(* PLC project Scenario_10, Beckhoff Automation GmbH TwinCAT PLC Control 3.5.8.40 *)
(* stored: creationDateTime 2017-05-02T11:08:00.4328535, modificationDateTime 2017-05-02T11:08:00.4378537 *)

PROGRAM MAIN
VAR		
	PPU : PPU;

//WPType	
	//Stack WPType
	Stack_WPType_Black : BOOL;
	Stack_WPType_White : BOOL;
	Stack_WPType_Metallic : BOOL;
	//Crane WPType
	Crane_WPType_Black : BOOL;
	Crane_WPType_White : BOOL;
	Crane_WPType_Metallic : BOOL;
	//Stamp WPType
	Stamp_WPType_Black : BOOL;
	Stamp_WPType_White : BOOL;
	Stamp_WPType_Metallic : BOOL;
	
//Free Signale for follow plant section
	//Stack
	Stack_WPProvided : BOOL;
	//Crane
	Crane_Allow_Conveyor_to_Operate : BOOL;
	Crane_Allow_Stamp_to_Operate : BOOL;
	Crane_PickedUpStackWP : BOOL;
	//Stamp	
	Stamp_IsStamping : BOOL;
	Stamp_WPAvailable : BOOL;
	Stamp_AutomaticExecuteCompleted	: BOOL;
	//Conveyor
	LargeSortingConveyor_AllowedToOperate : BOOL;
	LargeSortingConveyor_IsSorting : BOOL;
	LargeSortingConveyor_AutomaticExecuteCompleted : BOOL;
	
END_VAR

                  PPU();
PPU.Stack();
PPU.Crane();
PPU.Stamp();
PPU.LargeSortingConveyor();

//WPType
	//Stack WPType
	Stack_WPType_Black := PPU.Stack.WPType_Black;
	Stack_WPType_White := PPU.Stack.WPType_White;
	Stack_WPType_Metallic := PPU.Stack.WPType_Metallic;
	//Crane WPType
	Crane_WPType_Black := PPU.Crane.WPType_Black;
	Crane_WPType_White := PPU.Crane.WPType_White;
	Crane_WPType_Metallic := PPU.Crane.WPType_Metallic;
	//Stamp WPType
	Stamp_WPType_Black := PPU.Stamp.WPType_Black;
	Stamp_WPType_White := PPU.Stamp.WPType_White;
	Stamp_WPType_Metallic := PPU.Stamp.WPType_Metallic;
	
//Free Signale for follow plant section
	//Stack
	Stack_WPProvided := PPU.Stack.WPProvided;
	//Crane
	Crane_Allow_Conveyor_to_Operate := PPU.Crane.Conveyor_AllowedToOperate;
	Crane_Allow_Stamp_to_Operate := PPU.Crane.Stamp_AllowedToOperate;
	Crane_PickedUpStackWP := PPU.Crane.Table.AtStack.DI_SwitchTrue AND PPU.Crane.WPPickedUp;
	//Stamp
	Stamp_IsStamping := PPU.Stamp.IsStamping;
	Stamp_WPAvailable := PPU.Stamp.WPAvailable.DI_SwitchTrue;	
	Stamp_AutomaticExecuteCompleted := PPU.Stamp.AutomaticExecuteCompleted;
	//Conveyor
	LargeSortingConveyor_AllowedToOperate := Crane_Allow_Conveyor_to_Operate;
	LargeSortingConveyor_IsSorting := PPU.LargeSortingConveyor.IsSorting;
	LargeSortingConveyor_AutomaticExecuteCompleted := PPU.LargeSortingConveyor.AutomaticExecuteCompleted;
                
END_PROGRAM

FUNCTION_BLOCK BistableCylinder
VAR_INPUT	
END_VAR
VAR_OUTPUT
END_VAR
VAR	
	//Hardware
	DI_Extended AT %I* : BOOL;
	DI_Retracted AT %I* : BOOL;	
	DO_Extend AT %Q* : BOOL;
	DO_Retract AT %Q* : BOOL;
	//Software
	Extended : BOOL;
	Retracted : BOOL;
END_VAR

                  
                

ACTION ACT_Extend:
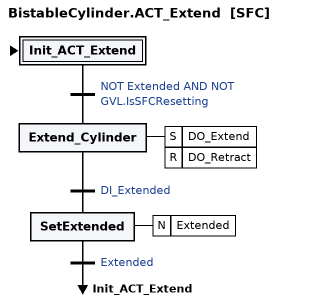
INITIAL_STEP Init_ACT_Extend:
END_STEP
TRANSITION FROM Init_ACT_Extend TO Extend_Cylinder
  := NOT Extended AND NOT GVL.IsSFCResetting;
END_TRANSITION
STEP Extend_Cylinder:
  DO_Extend(S);
  DO_Retract(R);
END_STEP
TRANSITION FROM Extend_Cylinder TO SetExtended
  := DI_Extended;
END_TRANSITION
STEP SetExtended:
  Extended(N);
END_STEP
TRANSITION FROM SetExtended TO Init_ACT_Extend
  := Extended;
END_TRANSITION
END_ACTION

ACTION ACT_Retract:
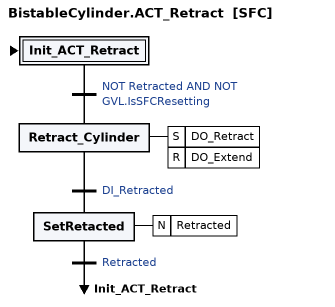
INITIAL_STEP Init_ACT_Retract:
END_STEP
TRANSITION FROM Init_ACT_Retract TO Retract_Cylinder
  := NOT Retracted AND NOT GVL.IsSFCResetting;
END_TRANSITION
STEP Retract_Cylinder:
  DO_Retract(S);
  DO_Extend(R);
END_STEP
TRANSITION FROM Retract_Cylinder TO SetRetacted
  := DI_Retracted;
END_TRANSITION
STEP SetRetacted:
  Retracted(N);
END_STEP
TRANSITION FROM SetRetacted TO Init_ACT_Retract
  := Retracted;
END_TRANSITION
END_ACTION
END_FUNCTION_BLOCK

FUNCTION_BLOCK InductiveSensor
VAR_INPUT
END_VAR
VAR_OUTPUT
END_VAR
VAR
	//Hardware
	DI_WPMetallic AT %I* : BOOL;
END_VAR

                  
                
END_FUNCTION_BLOCK

FUNCTION_BLOCK MicroSwitch
VAR_INPUT
END_VAR
VAR_OUTPUT
END_VAR
VAR
	//Hardware
	DI_SwitchTrue AT %I* : BOOL;
END_VAR

                  
                
END_FUNCTION_BLOCK

FUNCTION_BLOCK MonostableCylinder
VAR_INPUT	
END_VAR	
VAR_OUTPUT	
END_VAR
VAR	
	//Hardware
	DI_Extended AT %I* : BOOL;
	DI_Retracted AT %I* : BOOL;	
	DO_Extend AT %Q* : BOOL;
	//Software
	Extended : BOOL;
	Retracted : BOOL;
END_VAR

                  
                

ACTION ACT_Extend:
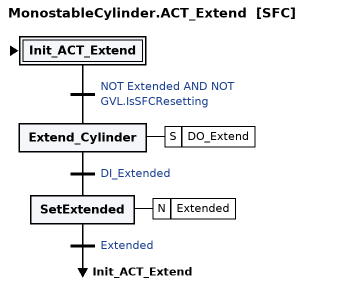
INITIAL_STEP Init_ACT_Extend:
END_STEP
TRANSITION FROM Init_ACT_Extend TO Extend_Cylinder
  := NOT Extended AND NOT GVL.IsSFCResetting;
END_TRANSITION
STEP Extend_Cylinder:
  DO_Extend(S);
END_STEP
TRANSITION FROM Extend_Cylinder TO SetExtended
  := DI_Extended;
END_TRANSITION
STEP SetExtended:
  Extended(N);
END_STEP
TRANSITION FROM SetExtended TO Init_ACT_Extend
  := Extended;
END_TRANSITION
END_ACTION

ACTION ACT_Retract:
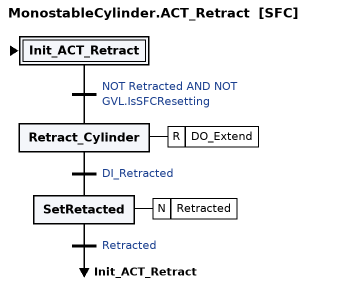
INITIAL_STEP Init_ACT_Retract:
END_STEP
TRANSITION FROM Init_ACT_Retract TO Retract_Cylinder
  := NOT Retracted AND NOT GVL.IsSFCResetting;
END_TRANSITION
STEP Retract_Cylinder:
  DO_Extend(R);
END_STEP
TRANSITION FROM Retract_Cylinder TO SetRetacted
  := DI_Retracted;
END_TRANSITION
STEP SetRetacted:
  Retracted(N);
END_STEP
TRANSITION FROM SetRetacted TO Init_ACT_Retract
  := Retracted;
END_TRANSITION
END_ACTION
END_FUNCTION_BLOCK

FUNCTION_BLOCK Motor
VAR_INPUT
END_VAR
VAR_OUTPUT	
END_VAR
VAR	
	//Hardware
	DO_TurnClockwise AT %Q* : BOOL;
	DO_TurnCounterclockwise AT %Q* : BOOL;
	//Software
	Stopped : BOOL;
	TurningClockwise : BOOL;
	TurningCounterclockwise : BOOL;
END_VAR

                  
                

ACTION ACT_Stop:
                      DO_TurnClockwise := FALSE;
DO_TurnCounterclockwise := FALSE;

Stopped := TRUE;
TurningClockwise := FALSE;
TurningCounterclockwise := FALSE;
                    
END_ACTION

ACTION ACT_TurnClockwise:
                      DO_TurnClockwise := TRUE;
DO_TurnCounterclockwise := FALSE;

Stopped := FALSE;
TurningClockwise := TRUE;
TurningCounterclockwise := FALSE;
                    
END_ACTION

ACTION ACT_TurnCounterclockwise:
                      DO_TurnClockwise := FALSE;
DO_TurnCounterclockwise := TRUE;

Stopped := FALSE;
TurningClockwise := FALSE;
TurningCounterclockwise := TRUE;
                    
END_ACTION
END_FUNCTION_BLOCK

FUNCTION_BLOCK OperationPanel
VAR_INPUT
END_VAR
VAR_OUTPUT
	//Software
	EmergencyStop : BOOL;
	StartButton : BOOL;
	ManuelMode : BOOL;
END_VAR
VAR
	//Hardware
	DI_StartButton AT %I* : BOOL;
	DI_ManuelButton AT %I* : BOOL;	
	DI_EmergencyStop AT %I* : BOOL;	
	DO_LampGreen AT %Q* : BOOL;
	DO_LampWhite AT %Q* : BOOL;
END_VAR

                  EmergencyStop := NOT DI_EmergencyStop;
StartButton := DI_StartButton;
ManuelMode := DI_ManuelButton;
                

ACTION ACT_TurnLampGreen_Off:
                      DO_LampGreen := FALSE;
                    
END_ACTION

ACTION ACT_TurnLampGreen_On:
                      DO_LampGreen := TRUE;
                    
END_ACTION

ACTION ACT_TurnLampWhite_Off:
                      DO_LampWhite:=FALSE;
                    
END_ACTION

ACTION ACT_TurnLampWhite_On:
                      DO_LampWhite:=TRUE;
                    
END_ACTION
END_FUNCTION_BLOCK

FUNCTION_BLOCK OpticalSensor
VAR_INPUT
END_VAR
VAR_OUTPUT
END_VAR
VAR
	//Hardware
	DI_WPLight AT %I* : BOOL;
END_VAR

                  
                
END_FUNCTION_BLOCK

FUNCTION_BLOCK PresenceSensor
VAR_INPUT
END_VAR
VAR_OUTPUT
END_VAR
VAR
	DI_WPDetected AT %I* : BOOL;
END_VAR

                  
                
END_FUNCTION_BLOCK

FUNCTION_BLOCK PressureSensor
VAR_INPUT
END_VAR
VAR_OUTPUT
END_VAR
VAR
	//Hardware
	AI_CurrentPressure AT %I* : INT;
END_VAR

                  
                
END_FUNCTION_BLOCK

FUNCTION_BLOCK ProportionalValve
VAR_INPUT
	//Hardware
	AO_SetPressure AT %Q* : INT;
END_VAR
VAR_OUTPUT
END_VAR
VAR	
END_VAR

                  
                
END_FUNCTION_BLOCK

FUNCTION_BLOCK TurningTable
VAR_INPUT
END_VAR
VAR_OUTPUT
END_VAR
VAR
	//Hardware
	Motor : Motor;
	AtStack : MicroSwitch;
	AtConveyor : MicroSwitch;
	AtStamp : MicroSwitch;
END_VAR

                  
                
END_FUNCTION_BLOCK

FUNCTION_BLOCK VacuumGripper
VAR_INPUT	
	//Hardware
	Valve : Valve;
	VacuumSwitch : VacuumSwitch;
END_VAR
VAR_OUTPUT	
END_VAR
VAR	
	//Software
	Intaken : BOOL;
	Released : BOOL;
END_VAR

                  
                

ACTION ACT_Intake:
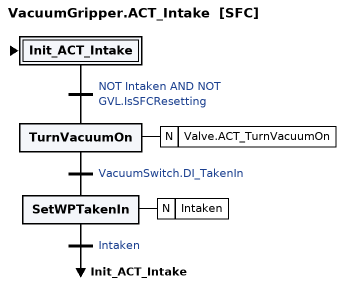
INITIAL_STEP Init_ACT_Intake:
END_STEP
TRANSITION FROM Init_ACT_Intake TO TurnVacuumOn
  := NOT Intaken AND NOT GVL.IsSFCResetting;
END_TRANSITION
STEP TurnVacuumOn:
  Valve.ACT_TurnVacuumOn(N);
END_STEP
TRANSITION FROM TurnVacuumOn TO SetWPTakenIn
  := VacuumSwitch.DI_TakenIn;
END_TRANSITION
STEP SetWPTakenIn:
  Intaken(N);
END_STEP
TRANSITION FROM SetWPTakenIn TO Init_ACT_Intake
  := Intaken;
END_TRANSITION
END_ACTION

ACTION ACT_Release:
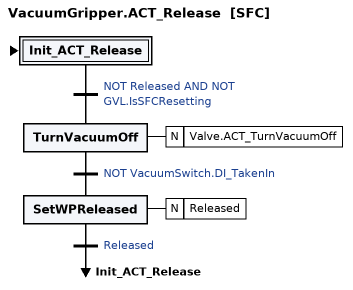
INITIAL_STEP Init_ACT_Release:
END_STEP
TRANSITION FROM Init_ACT_Release TO TurnVacuumOff
  := NOT Released AND NOT GVL.IsSFCResetting;
END_TRANSITION
STEP TurnVacuumOff:
  Valve.ACT_TurnVacuumOff(N);
END_STEP
TRANSITION FROM TurnVacuumOff TO SetWPReleased
  := NOT VacuumSwitch.DI_TakenIn;
END_TRANSITION
STEP SetWPReleased:
  Released(N);
END_STEP
TRANSITION FROM SetWPReleased TO Init_ACT_Release
  := Released;
END_TRANSITION
END_ACTION
END_FUNCTION_BLOCK

FUNCTION_BLOCK VacuumSwitch
VAR_INPUT
END_VAR
VAR_OUTPUT
END_VAR
VAR
	//Hardware
	DI_TakenIn AT %I* : BOOL;
END_VAR

                  
                
END_FUNCTION_BLOCK

FUNCTION_BLOCK Valve
VAR_INPUT
END_VAR
VAR_OUTPUT
END_VAR
VAR	
	//Hardware
	DO_VacuumOn AT %Q* : BOOL;
END_VAR

                  
                

ACTION ACT_TurnVacuumOff:
                      DO_VacuumOn := FALSE;
                    
END_ACTION

ACTION ACT_TurnVacuumOn:
                      DO_VacuumOn := TRUE;
                    
END_ACTION
END_FUNCTION_BLOCK

FUNCTION_BLOCK Crane
VAR_INPUT
	//Hardware
	LiftingCylinder : MonostableCylinder;
	Gripper : VacuumGripper;	
	Table : TurningTable;		
	//Software
	InitCompleted : BOOL;
	AutomaticExecuteCompleted : BOOL;			
	Conveyor_AllowedToOperate : BOOL;
	Stamp_AllowedToOperate : BOOL;
	Stamp_WPStamped : BOOL;
	SoftwareEmergency : BOOL;	
	EmergencyHandled : BOOL;
	SFCReset : BOOL;	//Only for SFC implementation
END_VAR
VAR_OUTPUT	
	//Software
	WPPickedUp : BOOL;
	WPPutDown : BOOL;
	ReachedStack : BOOL;
	ReachedConveyor : BOOL;
	ReachedStamp : BOOL;	
	WPType_White : BOOL;
	WPType_Black : BOOL;
	WPType_Metallic : BOOL;
END_VAR
VAR		
	//Hardware		
	CraneSpeed AT %Q* : INT;
	
	//Software
	Timer : TON;
	Check_Stack_WPProvided : BOOL;
	Check_Stack_WPType_Black : BOOL;
	Check_Stack_WPType_White : BOOL;
	Check_Stack_WPType_Metallic : BOOL;
	Check_LargeSortingConveyor_IsSorting : BOOL;
	Check_LargeSortingConveyor_AutomaticExecuteCompleted :BOOL;	
	Check_Stamp_IsStamping : BOOL;
	Check_Stamp_WPAvailable : BOOL;
	Check_Stamp_AutomaticExecuteCompleted : BOOL;
END_VAR

                  Check_Stack_WPProvided := Main.Stack_WPProvided;
Check_Stack_WPType_Black := Main.Stack_WPType_Black;
Check_Stack_WPType_White := Main.Stack_WPType_White;
Check_Stack_WPType_Metallic := Main.Stack_WPType_Metallic;
Check_LargeSortingConveyor_IsSorting := Main.LargeSortingConveyor_IsSorting;
Check_LargeSortingConveyor_AutomaticExecuteCompleted := Main.LargeSortingConveyor_AutomaticExecuteCompleted;
Check_Stamp_IsStamping := Main.Stamp_IsStamping;
Check_Stamp_WPAvailable := Main.Stamp_WPAvailable;
Check_Stamp_AutomaticExecuteCompleted := Main.Stamp_AutomaticExecuteCompleted;

                

ACTION Reset_ConveyorAllowedToOperate:
                      Conveyor_AllowedToOperate := FALSE;
                    
END_ACTION

ACTION Reset_StampAllowedToOperate:
                      Stamp_AllowedToOperate := FALSE;
                    
END_ACTION

ACTION Reset_Timer:
                      Timer(IN:=FALSE);
                    
END_ACTION

ACTION Reset_Variables:
                      InitCompleted := FALSE;
AutomaticExecuteCompleted := FALSE;
Conveyor_AllowedToOperate := FALSE;
Stamp_AllowedToOperate := FALSE;

WPPickedUp := FALSE;
WPPutDown := FALSE;
ReachedStack := FALSE;
ReachedConveyor := FALSE;
ReachedStamp := FALSE;	
WPType_White := FALSE;
WPType_Black := FALSE;
WPType_Metallic := FALSE;
                    
END_ACTION

ACTION Set_ConveyorAllowedToOperate:
                      Conveyor_AllowedToOperate := TRUE;
                    
END_ACTION

ACTION Set_StampAllowedToOperate:
                      Stamp_AllowedToOperate := TRUE;
                    
END_ACTION

ACTION Set_Timer50ms:
                      Timer(IN:=TRUE, PT:=T#50MS);
                    
END_ACTION

ACTION Set_WPTypeEqualsStack:
                      WPType_White:=Main.Stack_WPType_White;
WPType_Black:=Main.Stack_WPType_Black;	
WPType_Metallic:=Main.Stack_WPType_Metallic;
                    
END_ACTION

ACTION Set_WPTypeEqualsStamp:
                      WPType_White:=Main.Stamp_WPType_White;
WPType_Black:=Main.Stamp_WPType_Black;	
WPType_Metallic:=Main.Stamp_WPType_Metallic;
                    
END_ACTION

ACTION TurnClockwise_AND_Timer8000ms:
                      Table.Motor.ACT_TurnClockwise();
Timer(IN:=TRUE, PT:=T#8000MS);
                    
END_ACTION

ACTION TurnCounterclockwise_AND_Timer8000ms:
                      Table.Motor.ACT_TurnCounterclockwise();
Timer(IN:=TRUE, PT:=T#8000MS);
                    
END_ACTION

ACTION TurnVacuumOn_AND_Timer2000ms:
                      Gripper.ACT_Intake();
Timer(IN:=TRUE, PT:=T#2000MS);
                    
END_ACTION

ACTION ACT_MoveToConveyor:
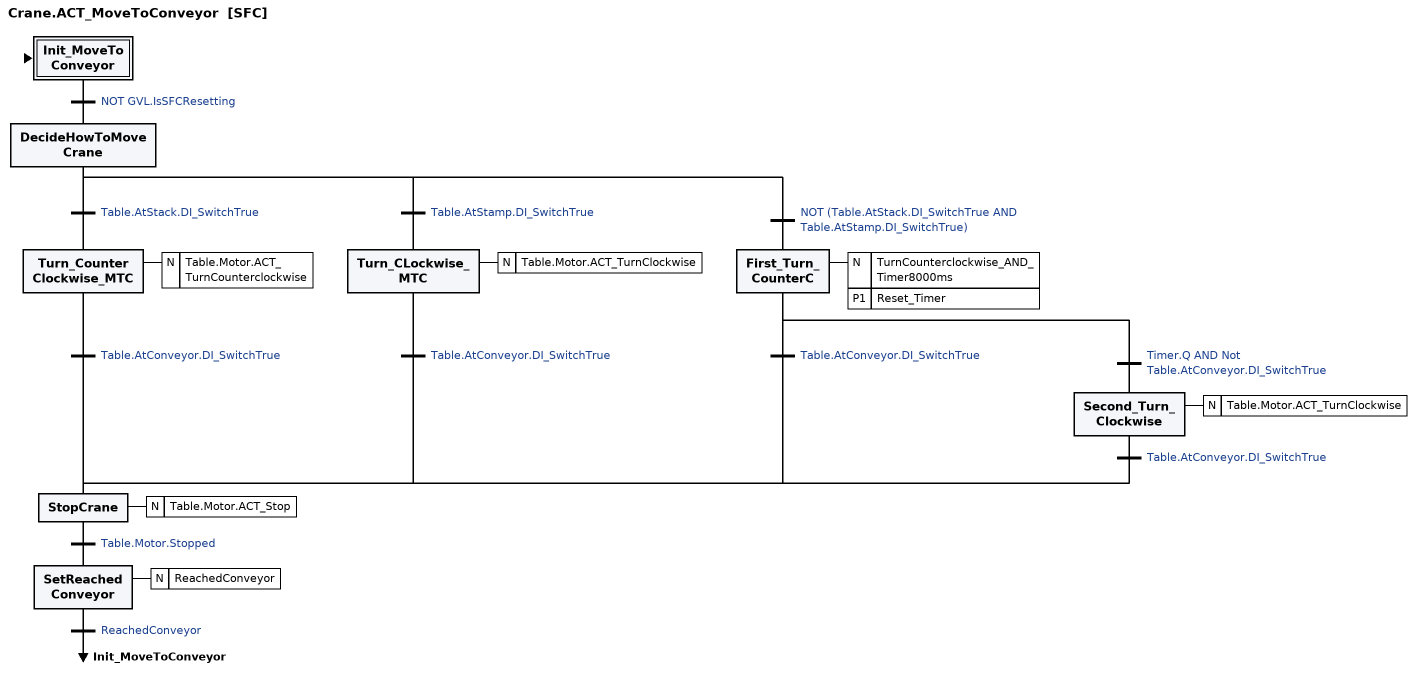
INITIAL_STEP Init_MoveToConveyor:
END_STEP
TRANSITION FROM Init_MoveToConveyor TO DecideHowToMoveCrane
  := NOT GVL.IsSFCResetting;
END_TRANSITION
STEP DecideHowToMoveCrane:
END_STEP
TRANSITION FROM DecideHowToMoveCrane TO Turn_CounterClockwise_MTC
  := Table.AtStack.DI_SwitchTrue;
END_TRANSITION
TRANSITION FROM DecideHowToMoveCrane TO Turn_CLockwise_MTC
  := Table.AtStamp.DI_SwitchTrue;
END_TRANSITION
TRANSITION FROM DecideHowToMoveCrane TO First_Turn_CounterC
  := NOT (Table.AtStack.DI_SwitchTrue AND Table.AtStamp.DI_SwitchTrue);
END_TRANSITION
STEP Turn_CounterClockwise_MTC:
  Table.Motor.ACT_TurnCounterclockwise(N);
END_STEP
TRANSITION FROM Turn_CounterClockwise_MTC TO StopCrane
  := Table.AtConveyor.DI_SwitchTrue;
END_TRANSITION
STEP Turn_CLockwise_MTC:
  Table.Motor.ACT_TurnClockwise(N);
END_STEP
TRANSITION FROM Turn_CLockwise_MTC TO StopCrane
  := Table.AtConveyor.DI_SwitchTrue;
END_TRANSITION
STEP First_Turn_CounterC:
  TurnCounterclockwise_AND_Timer8000ms(N);
  Reset_Timer(P1);
END_STEP
TRANSITION FROM First_Turn_CounterC TO StopCrane
  := Table.AtConveyor.DI_SwitchTrue;
END_TRANSITION
TRANSITION FROM First_Turn_CounterC TO Second_Turn_Clockwise
  := Timer.Q AND Not Table.AtConveyor.DI_SwitchTrue;
END_TRANSITION
STEP Second_Turn_Clockwise:
  Table.Motor.ACT_TurnClockwise(N);
END_STEP
TRANSITION FROM Second_Turn_Clockwise TO StopCrane
  := Table.AtConveyor.DI_SwitchTrue;
END_TRANSITION
STEP StopCrane:
  Table.Motor.ACT_Stop(N);
END_STEP
TRANSITION FROM StopCrane TO SetReachedConveyor
  := Table.Motor.Stopped;
END_TRANSITION
STEP SetReachedConveyor:
  ReachedConveyor(N);
END_STEP
TRANSITION FROM SetReachedConveyor TO Init_MoveToConveyor
  := ReachedConveyor;
END_TRANSITION
END_ACTION

ACTION ACT_MoveToStack:
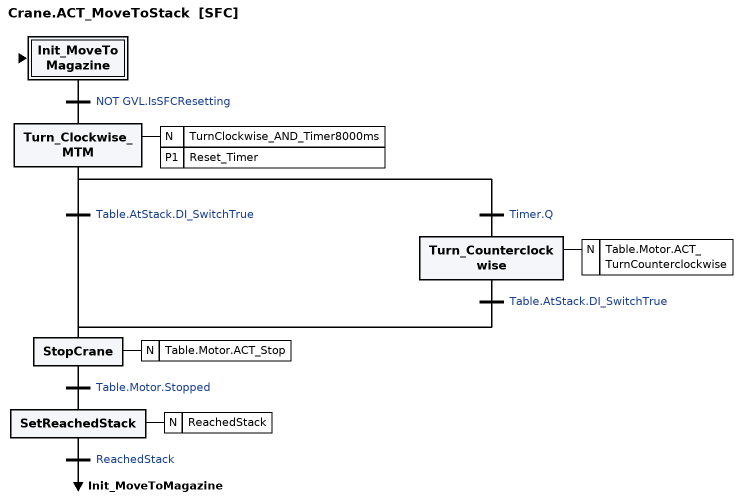
INITIAL_STEP Init_MoveToMagazine:
END_STEP
TRANSITION FROM Init_MoveToMagazine TO Turn_Clockwise_MTM
  := NOT GVL.IsSFCResetting;
END_TRANSITION
STEP Turn_Clockwise_MTM:
  TurnClockwise_AND_Timer8000ms(N);
  Reset_Timer(P1);
END_STEP
TRANSITION FROM Turn_Clockwise_MTM TO StopCrane
  := Table.AtStack.DI_SwitchTrue;
END_TRANSITION
TRANSITION FROM Turn_Clockwise_MTM TO Turn_Counterclockwise
  := Timer.Q;
END_TRANSITION
STEP Turn_Counterclockwise:
  Table.Motor.ACT_TurnCounterclockwise(N);
END_STEP
TRANSITION FROM Turn_Counterclockwise TO StopCrane
  := Table.AtStack.DI_SwitchTrue;
END_TRANSITION
STEP StopCrane:
  Table.Motor.ACT_Stop(N);
END_STEP
TRANSITION FROM StopCrane TO SetReachedStack
  := Table.Motor.Stopped;
END_TRANSITION
STEP SetReachedStack:
  ReachedStack(N);
END_STEP
TRANSITION FROM SetReachedStack TO Init_MoveToMagazine
  := ReachedStack;
END_TRANSITION
END_ACTION

ACTION ACT_MoveToStamp:
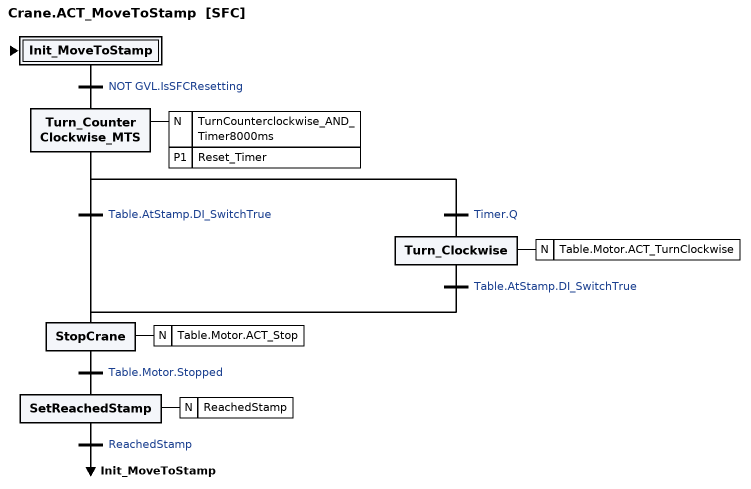
INITIAL_STEP Init_MoveToStamp:
END_STEP
TRANSITION FROM Init_MoveToStamp TO Turn_CounterClockwise_MTS
  := NOT GVL.IsSFCResetting;
END_TRANSITION
STEP Turn_CounterClockwise_MTS:
  TurnCounterclockwise_AND_Timer8000ms(N);
  Reset_Timer(P1);
END_STEP
TRANSITION FROM Turn_CounterClockwise_MTS TO StopCrane
  := Table.AtStamp.DI_SwitchTrue;
END_TRANSITION
TRANSITION FROM Turn_CounterClockwise_MTS TO Turn_Clockwise
  := Timer.Q;
END_TRANSITION
STEP Turn_Clockwise:
  Table.Motor.ACT_TurnClockwise(N);
END_STEP
TRANSITION FROM Turn_Clockwise TO StopCrane
  := Table.AtStamp.DI_SwitchTrue;
END_TRANSITION
STEP StopCrane:
  Table.Motor.ACT_Stop(N);
END_STEP
TRANSITION FROM StopCrane TO SetReachedStamp
  := Table.Motor.Stopped;
END_TRANSITION
STEP SetReachedStamp:
  ReachedStamp(N);
END_STEP
TRANSITION FROM SetReachedStamp TO Init_MoveToStamp
  := ReachedStamp;
END_TRANSITION
END_ACTION

ACTION ACT_PickUpWP:
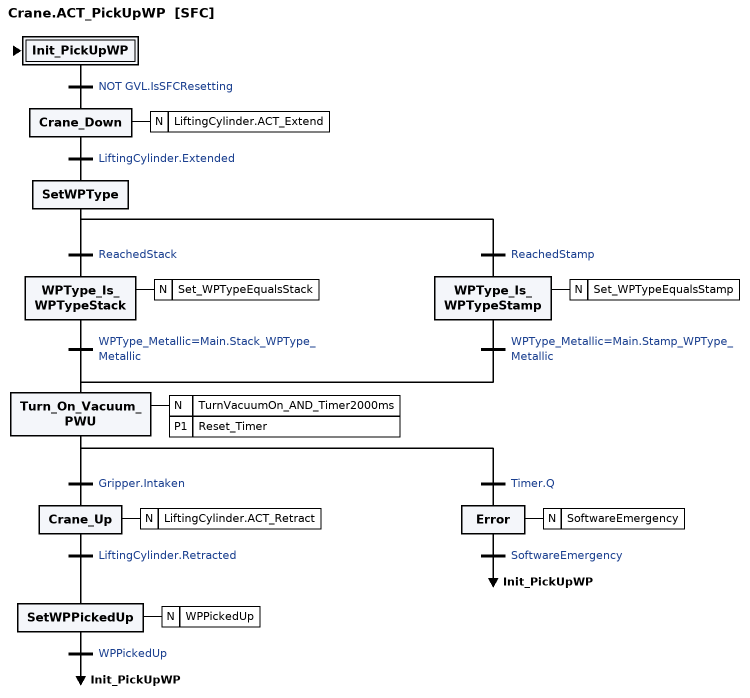
INITIAL_STEP Init_PickUpWP:
END_STEP
TRANSITION FROM Init_PickUpWP TO Crane_Down
  := NOT GVL.IsSFCResetting;
END_TRANSITION
STEP Crane_Down:
  LiftingCylinder.ACT_Extend(N);
END_STEP
TRANSITION FROM Crane_Down TO SetWPType
  := LiftingCylinder.Extended;
END_TRANSITION
STEP SetWPType:
END_STEP
TRANSITION FROM SetWPType TO WPType_Is_WPTypeStack
  := ReachedStack;
END_TRANSITION
TRANSITION FROM SetWPType TO WPType_Is_WPTypeStamp
  := ReachedStamp;
END_TRANSITION
STEP WPType_Is_WPTypeStack:
  Set_WPTypeEqualsStack(N);
END_STEP
TRANSITION FROM WPType_Is_WPTypeStack TO Turn_On_Vacuum_PWU
  := WPType_Metallic=Main.Stack_WPType_Metallic;
END_TRANSITION
STEP WPType_Is_WPTypeStamp:
  Set_WPTypeEqualsStamp(N);
END_STEP
TRANSITION FROM WPType_Is_WPTypeStamp TO Turn_On_Vacuum_PWU
  := WPType_Metallic=Main.Stamp_WPType_Metallic;
END_TRANSITION
STEP Turn_On_Vacuum_PWU:
  TurnVacuumOn_AND_Timer2000ms(N);
  Reset_Timer(P1);
END_STEP
TRANSITION FROM Turn_On_Vacuum_PWU TO Crane_Up
  := Gripper.Intaken;
END_TRANSITION
TRANSITION FROM Turn_On_Vacuum_PWU TO Error
  := Timer.Q;
END_TRANSITION
STEP Crane_Up:
  LiftingCylinder.ACT_Retract(N);
END_STEP
TRANSITION FROM Crane_Up TO SetWPPickedUp
  := LiftingCylinder.Retracted;
END_TRANSITION
STEP Error:
  SoftwareEmergency(N);
END_STEP
TRANSITION FROM Error TO Init_PickUpWP
  := SoftwareEmergency;
END_TRANSITION
STEP SetWPPickedUp:
  WPPickedUp(N);
END_STEP
TRANSITION FROM SetWPPickedUp TO Init_PickUpWP
  := WPPickedUp;
END_TRANSITION
END_ACTION

ACTION ACT_PutDownWP:
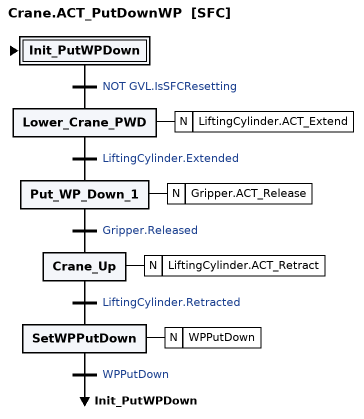
INITIAL_STEP Init_PutWPDown:
END_STEP
TRANSITION FROM Init_PutWPDown TO Lower_Crane_PWD
  := NOT GVL.IsSFCResetting;
END_TRANSITION
STEP Lower_Crane_PWD:
  LiftingCylinder.ACT_Extend(N);
END_STEP
TRANSITION FROM Lower_Crane_PWD TO Put_WP_Down_1
  := LiftingCylinder.Extended;
END_TRANSITION
STEP Put_WP_Down_1:
  Gripper.ACT_Release(N);
END_STEP
TRANSITION FROM Put_WP_Down_1 TO Crane_Up
  := Gripper.Released;
END_TRANSITION
STEP Crane_Up:
  LiftingCylinder.ACT_Retract(N);
END_STEP
TRANSITION FROM Crane_Up TO SetWPPutDown
  := LiftingCylinder.Retracted;
END_TRANSITION
STEP SetWPPutDown:
  WPPutDown(N);
END_STEP
TRANSITION FROM SetWPPutDown TO Init_PutWPDown
  := WPPutDown;
END_TRANSITION
END_ACTION

ACTION ACT_AutomaticExecute:
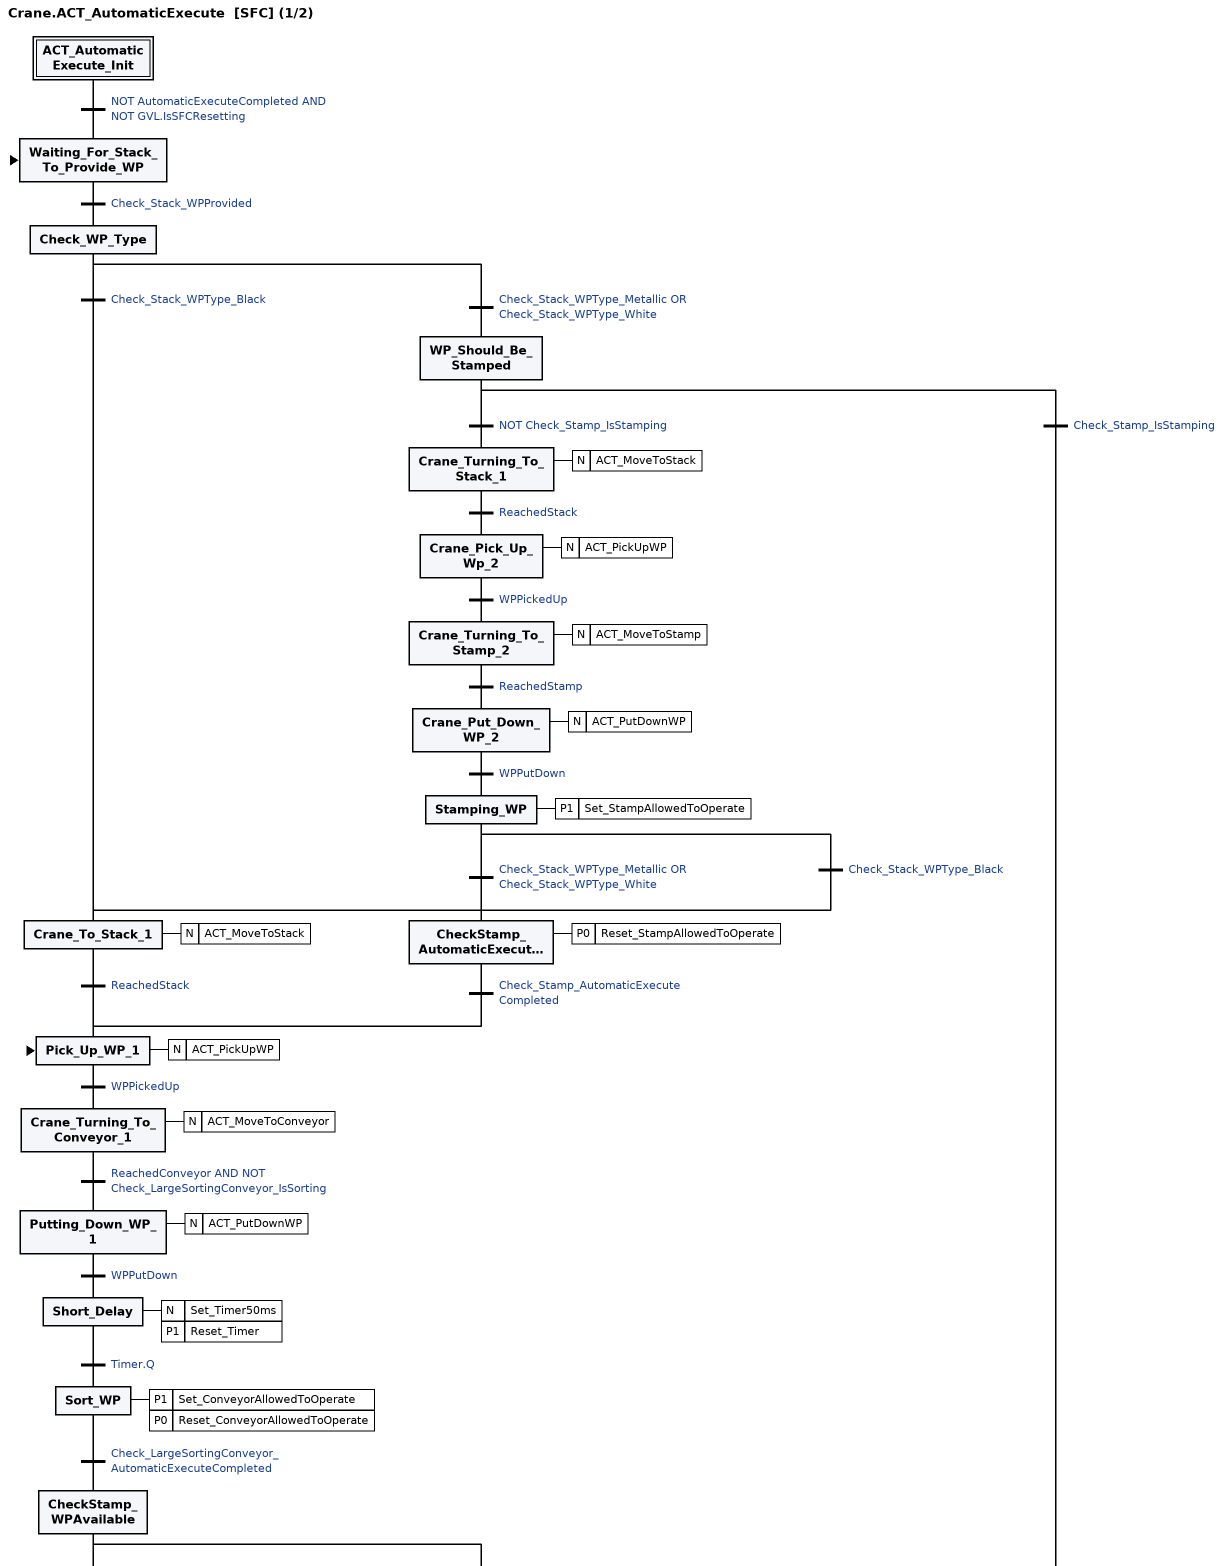
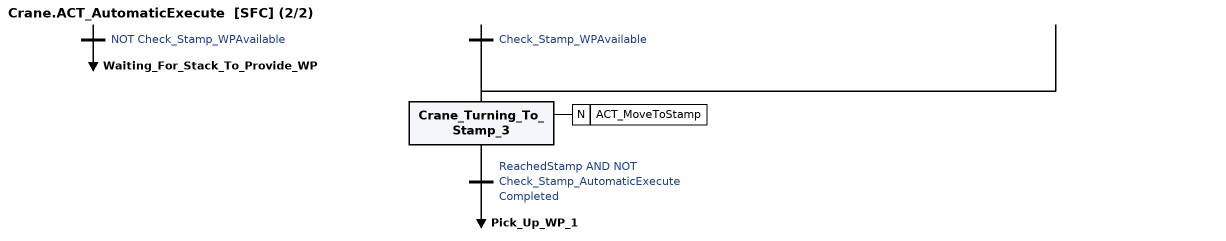
INITIAL_STEP ACT_AutomaticExecute_Init:
END_STEP
TRANSITION FROM ACT_AutomaticExecute_Init TO Waiting_For_Stack_To_Provide_WP
  := NOT AutomaticExecuteCompleted AND NOT GVL.IsSFCResetting;
END_TRANSITION
STEP Waiting_For_Stack_To_Provide_WP:
END_STEP
TRANSITION FROM Waiting_For_Stack_To_Provide_WP TO Check_WP_Type
  := Check_Stack_WPProvided;
END_TRANSITION
STEP Check_WP_Type:
END_STEP
TRANSITION FROM Check_WP_Type TO Crane_To_Stack_1
  := Check_Stack_WPType_Black;
END_TRANSITION
TRANSITION FROM Check_WP_Type TO WP_Should_Be_Stamped
  := Check_Stack_WPType_Metallic OR Check_Stack_WPType_White;
END_TRANSITION
STEP Crane_To_Stack_1:
  ACT_MoveToStack(N);
END_STEP
TRANSITION FROM Crane_To_Stack_1 TO Pick_Up_WP_1
  := ReachedStack;
END_TRANSITION
STEP Pick_Up_WP_1:
  ACT_PickUpWP(N);
END_STEP
TRANSITION FROM Pick_Up_WP_1 TO Crane_Turning_To_Conveyor_1
  := WPPickedUp;
END_TRANSITION
STEP Crane_Turning_To_Conveyor_1:
  ACT_MoveToConveyor(N);
END_STEP
TRANSITION FROM Crane_Turning_To_Conveyor_1 TO Putting_Down_WP_1
  := ReachedConveyor AND NOT Check_LargeSortingConveyor_IsSorting;
END_TRANSITION
STEP Putting_Down_WP_1:
  ACT_PutDownWP(N);
END_STEP
TRANSITION FROM Putting_Down_WP_1 TO Short_Delay
  := WPPutDown;
END_TRANSITION
STEP Short_Delay:
  Set_Timer50ms(N);
  Reset_Timer(P1);
END_STEP
TRANSITION FROM Short_Delay TO Sort_WP
  := Timer.Q;
END_TRANSITION
STEP Sort_WP:
  Set_ConveyorAllowedToOperate(P1);
  Reset_ConveyorAllowedToOperate(P0);
END_STEP
TRANSITION FROM Sort_WP TO CheckStamp_WPAvailable
  := Check_LargeSortingConveyor_AutomaticExecuteCompleted;
END_TRANSITION
STEP CheckStamp_WPAvailable:
END_STEP
TRANSITION FROM CheckStamp_WPAvailable TO Waiting_For_Stack_To_Provide_WP
  := NOT Check_Stamp_WPAvailable;
END_TRANSITION
TRANSITION FROM CheckStamp_WPAvailable TO Crane_Turning_To_Stamp_3
  := Check_Stamp_WPAvailable;
END_TRANSITION
STEP WP_Should_Be_Stamped:
END_STEP
TRANSITION FROM WP_Should_Be_Stamped TO Crane_Turning_To_Stack_1
  := NOT Check_Stamp_IsStamping;
END_TRANSITION
TRANSITION FROM WP_Should_Be_Stamped TO Crane_Turning_To_Stamp_3
  := Check_Stamp_IsStamping;
END_TRANSITION
STEP Crane_Turning_To_Stack_1:
  ACT_MoveToStack(N);
END_STEP
TRANSITION FROM Crane_Turning_To_Stack_1 TO Crane_Pick_Up_Wp_2
  := ReachedStack;
END_TRANSITION
STEP Crane_Pick_Up_Wp_2:
  ACT_PickUpWP(N);
END_STEP
TRANSITION FROM Crane_Pick_Up_Wp_2 TO Crane_Turning_To_Stamp_2
  := WPPickedUp;
END_TRANSITION
STEP Crane_Turning_To_Stamp_2:
  ACT_MoveToStamp(N);
END_STEP
TRANSITION FROM Crane_Turning_To_Stamp_2 TO Crane_Put_Down_WP_2
  := ReachedStamp;
END_TRANSITION
STEP Crane_Put_Down_WP_2:
  ACT_PutDownWP(N);
END_STEP
TRANSITION FROM Crane_Put_Down_WP_2 TO Stamping_WP
  := WPPutDown;
END_TRANSITION
STEP Stamping_WP:
  Set_StampAllowedToOperate(P1);
END_STEP
TRANSITION FROM Stamping_WP TO CheckStamp_AutomaticExecuteCompleted
  := Check_Stack_WPType_Metallic OR Check_Stack_WPType_White;
END_TRANSITION
TRANSITION FROM Stamping_WP TO Crane_To_Stack_1
  := Check_Stack_WPType_Black;
END_TRANSITION
STEP CheckStamp_AutomaticExecuteCompleted:
  Reset_StampAllowedToOperate(P0);
END_STEP
TRANSITION FROM CheckStamp_AutomaticExecuteCompleted TO Pick_Up_WP_1
  := Check_Stamp_AutomaticExecuteCompleted;
END_TRANSITION
STEP Crane_Turning_To_Stamp_3:
  ACT_MoveToStamp(N);
END_STEP
TRANSITION FROM Crane_Turning_To_Stamp_3 TO Pick_Up_WP_1
  := ReachedStamp AND NOT Check_Stamp_AutomaticExecuteCompleted;
END_TRANSITION
END_ACTION

ACTION ACT_EmergencyStop:
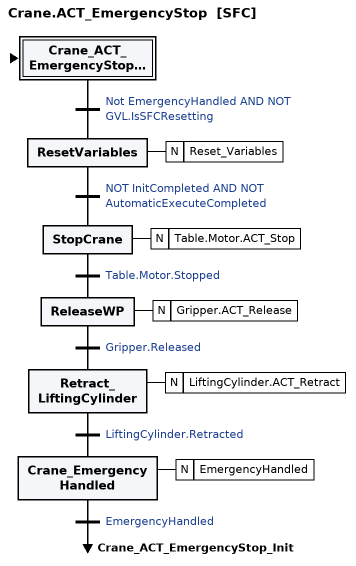
INITIAL_STEP Crane_ACT_EmergencyStop_Init:
END_STEP
TRANSITION FROM Crane_ACT_EmergencyStop_Init TO ResetVariables
  := Not EmergencyHandled AND NOT GVL.IsSFCResetting;
END_TRANSITION
STEP ResetVariables:
  Reset_Variables(N);
END_STEP
TRANSITION FROM ResetVariables TO StopCrane
  := NOT InitCompleted AND NOT AutomaticExecuteCompleted;
END_TRANSITION
STEP StopCrane:
  Table.Motor.ACT_Stop(N);
END_STEP
TRANSITION FROM StopCrane TO ReleaseWP
  := Table.Motor.Stopped;
END_TRANSITION
STEP ReleaseWP:
  Gripper.ACT_Release(N);
END_STEP
TRANSITION FROM ReleaseWP TO Retract_LiftingCylinder
  := Gripper.Released;
END_TRANSITION
STEP Retract_LiftingCylinder:
  LiftingCylinder.ACT_Retract(N);
END_STEP
TRANSITION FROM Retract_LiftingCylinder TO Crane_EmergencyHandled
  := LiftingCylinder.Retracted;
END_TRANSITION
STEP Crane_EmergencyHandled:
  EmergencyHandled(N);
END_STEP
TRANSITION FROM Crane_EmergencyHandled TO Crane_ACT_EmergencyStop_Init
  := EmergencyHandled;
END_TRANSITION
END_ACTION

ACTION ACT_Init:
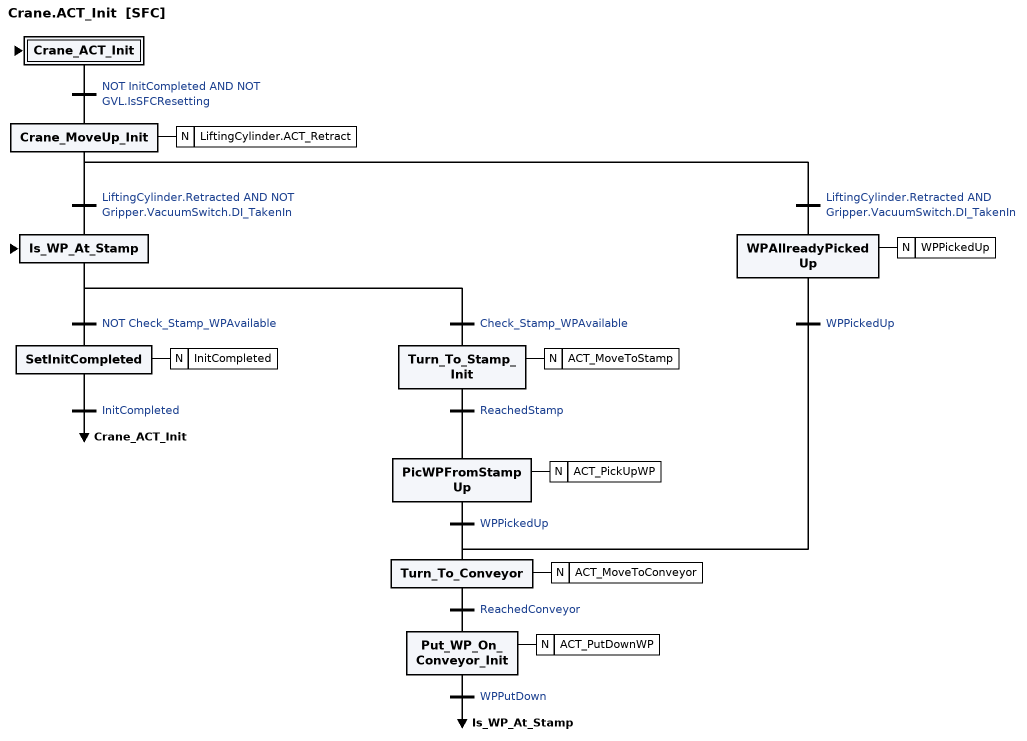
INITIAL_STEP Crane_ACT_Init:
END_STEP
TRANSITION FROM Crane_ACT_Init TO Crane_MoveUp_Init
  := NOT InitCompleted AND NOT GVL.IsSFCResetting;
END_TRANSITION
STEP Crane_MoveUp_Init:
  LiftingCylinder.ACT_Retract(N);
END_STEP
TRANSITION FROM Crane_MoveUp_Init TO Is_WP_At_Stamp
  := LiftingCylinder.Retracted AND NOT Gripper.VacuumSwitch.DI_TakenIn;
END_TRANSITION
TRANSITION FROM Crane_MoveUp_Init TO WPAllreadyPickedUp
  := LiftingCylinder.Retracted AND Gripper.VacuumSwitch.DI_TakenIn;
END_TRANSITION
STEP WPAllreadyPickedUp:
  WPPickedUp(N);
END_STEP
TRANSITION FROM WPAllreadyPickedUp TO Turn_To_Conveyor
  := WPPickedUp;
END_TRANSITION
STEP Turn_To_Conveyor:
  ACT_MoveToConveyor(N);
END_STEP
TRANSITION FROM Turn_To_Conveyor TO Put_WP_On_Conveyor_Init
  := ReachedConveyor;
END_TRANSITION
STEP Put_WP_On_Conveyor_Init:
  ACT_PutDownWP(N);
END_STEP
TRANSITION FROM Put_WP_On_Conveyor_Init TO Is_WP_At_Stamp
  := WPPutDown;
END_TRANSITION
STEP Is_WP_At_Stamp:
END_STEP
TRANSITION FROM Is_WP_At_Stamp TO SetInitCompleted
  := NOT Check_Stamp_WPAvailable;
END_TRANSITION
TRANSITION FROM Is_WP_At_Stamp TO Turn_To_Stamp_Init
  := Check_Stamp_WPAvailable;
END_TRANSITION
STEP Turn_To_Stamp_Init:
  ACT_MoveToStamp(N);
END_STEP
TRANSITION FROM Turn_To_Stamp_Init TO PicWPFromStampUp
  := ReachedStamp;
END_TRANSITION
STEP PicWPFromStampUp:
  ACT_PickUpWP(N);
END_STEP
TRANSITION FROM PicWPFromStampUp TO Turn_To_Conveyor
  := WPPickedUp;
END_TRANSITION
STEP SetInitCompleted:
  InitCompleted(N);
END_STEP
TRANSITION FROM SetInitCompleted TO Crane_ACT_Init
  := InitCompleted;
END_TRANSITION
END_ACTION
END_FUNCTION_BLOCK

FUNCTION_BLOCK LargeSortingConveyor
VAR_INPUT
	//Hardware
	Panel : OperationPanel;	
	Motor : Motor;
	Seperator1 : MonostableCylinder;
	Seperator2 : MonostableCylinder;	
	PsBeginning : PresenceSensor;		
	OptRamp1 : OpticalSensor;
	IndRamp1 : InductiveSensor;
	OptRamp2 : OpticalSensor;
	IndRamp2 : InductiveSensor;
	OptEnd : OpticalSensor;	
	
	Check_Allowed_To_Operate : BOOL;
	SFCReset : BOOL;	//Only for SFC implementation
END_VAR
VAR_OUTPUT	
	//Software	
	StartButton : BOOL;
	InitCompleted : BOOL;
	AutomaticExecuteCompleted : BOOL;
	EmergencyStop : BOOL;
	EmergencyHandled : BOOL;	
	IsSorting : BOOL;		
END_VAR
VAR	
	//Hardware		
	ConveyorSpeed AT %Q* : INT;

	//Software
	WPSorted : BOOL;
	WPTypeChecked : BOOL;
	TargetChanged : BOOL;	
	WPType_White : BOOL;
	WPType_Black : BOOL;
	WPType_Metallic : BOOL;
	CurrentTarget_Ramp1 : BOOL;
	CurrentTarget_Ramp2 : BOOL;
	CurrentTarget_Ramp3 : BOOL;	
	Priority_White : INT;
	Priority_Black: INT;
	Priority_Metallic : INT;
	CounterVar : INT;
END_VAR

                  Panel();
StartButton := Panel.StartButton;
EmergencyStop := Panel.EmergencyStop;
Check_Allowed_To_Operate := Main.Crane_Allow_Conveyor_to_Operate;
                

ACTION Reset_Variables:
                      InitCompleted := FALSE;
AutomaticExecuteCompleted := FALSE;

WPSorted:=FALSE;
IsSorting:=FALSE;
WPTypeChecked:=FALSE;
TargetChanged:=FALSE;
WPType_White:=FALSE;
WPType_Black:=FALSE;
WPType_Metallic:=FALSE;
CurrentTarget_Ramp1:=FALSE;
CurrentTarget_Ramp2:=FALSE;
CurrentTarget_Ramp3:=FALSE;
                    
END_ACTION

ACTION SelectRamp:
                      CounterVar := CounterVar MOD 10;
CounterVar := CounterVar + 1;
                    
END_ACTION

ACTION Set_PriorityBlack:
                      Priority_Black := 1;
                    
END_ACTION

ACTION Set_PriorityMetallic:
                      Priority_Metallic := 1;
                    
END_ACTION

ACTION Set_PriorityWhite:
                      Priority_White := 1;
                    
END_ACTION

ACTION ACT_ChangeTarget:
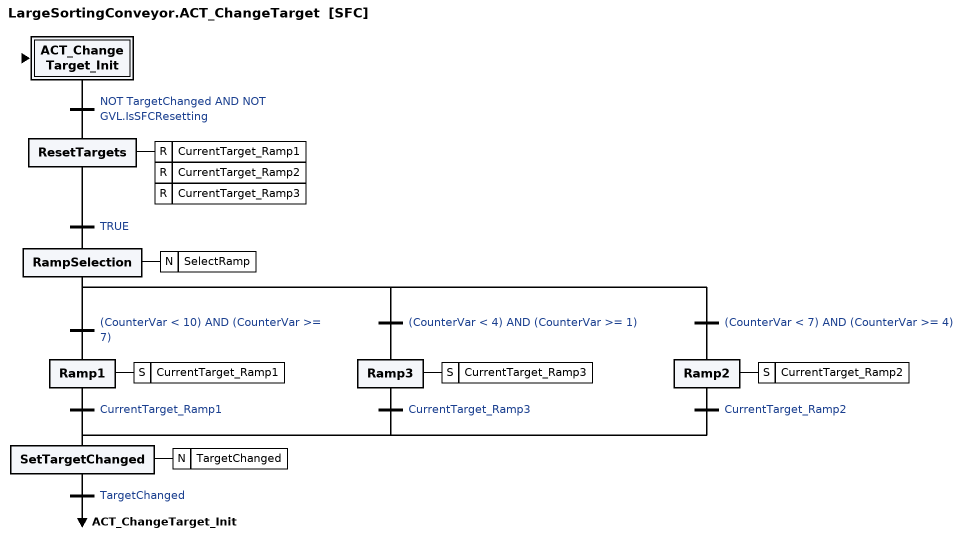
INITIAL_STEP ACT_ChangeTarget_Init:
END_STEP
TRANSITION FROM ACT_ChangeTarget_Init TO ResetTargets
  := NOT TargetChanged AND NOT GVL.IsSFCResetting;
END_TRANSITION
STEP ResetTargets:
  CurrentTarget_Ramp1(R);
  CurrentTarget_Ramp2(R);
  CurrentTarget_Ramp3(R);
END_STEP
TRANSITION FROM ResetTargets TO RampSelection
  := TRUE;
END_TRANSITION
STEP RampSelection:
  SelectRamp(N);
END_STEP
TRANSITION FROM RampSelection TO Ramp1
  := (CounterVar < 10) AND (CounterVar >= 7);
END_TRANSITION
TRANSITION FROM RampSelection TO Ramp3
  := (CounterVar < 4) AND (CounterVar >= 1);
END_TRANSITION
TRANSITION FROM RampSelection TO Ramp2
  := (CounterVar < 7) AND (CounterVar >= 4);
END_TRANSITION
STEP Ramp1:
  CurrentTarget_Ramp1(S);
END_STEP
TRANSITION FROM Ramp1 TO SetTargetChanged
  := CurrentTarget_Ramp1;
END_TRANSITION
STEP Ramp3:
  CurrentTarget_Ramp3(S);
END_STEP
TRANSITION FROM Ramp3 TO SetTargetChanged
  := CurrentTarget_Ramp3;
END_TRANSITION
STEP Ramp2:
  CurrentTarget_Ramp2(S);
END_STEP
TRANSITION FROM Ramp2 TO SetTargetChanged
  := CurrentTarget_Ramp2;
END_TRANSITION
STEP SetTargetChanged:
  TargetChanged(N);
END_STEP
TRANSITION FROM SetTargetChanged TO ACT_ChangeTarget_Init
  := TargetChanged;
END_TRANSITION
END_ACTION

ACTION ACT_CheckWPType:
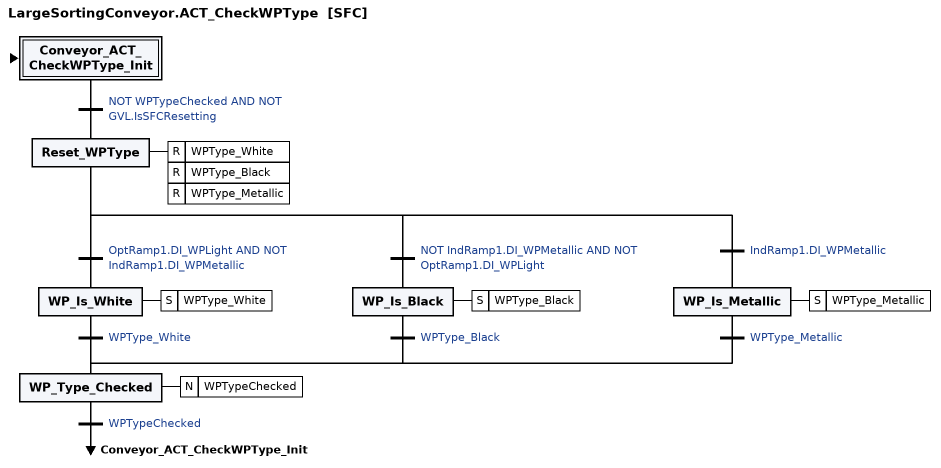
INITIAL_STEP Conveyor_ACT_CheckWPType_Init:
END_STEP
TRANSITION FROM Conveyor_ACT_CheckWPType_Init TO Reset_WPType
  := NOT WPTypeChecked AND NOT GVL.IsSFCResetting;
END_TRANSITION
STEP Reset_WPType:
  WPType_White(R);
  WPType_Black(R);
  WPType_Metallic(R);
END_STEP
TRANSITION FROM Reset_WPType TO WP_Is_White
  := OptRamp1.DI_WPLight AND NOT IndRamp1.DI_WPMetallic;
END_TRANSITION
TRANSITION FROM Reset_WPType TO WP_Is_Black
  := NOT IndRamp1.DI_WPMetallic AND NOT OptRamp1.DI_WPLight;
END_TRANSITION
TRANSITION FROM Reset_WPType TO WP_Is_Metallic
  := IndRamp1.DI_WPMetallic;
END_TRANSITION
STEP WP_Is_White:
  WPType_White(S);
END_STEP
TRANSITION FROM WP_Is_White TO WP_Type_Checked
  := WPType_White;
END_TRANSITION
STEP WP_Is_Black:
  WPType_Black(S);
END_STEP
TRANSITION FROM WP_Is_Black TO WP_Type_Checked
  := WPType_Black;
END_TRANSITION
STEP WP_Is_Metallic:
  WPType_Metallic(S);
END_STEP
TRANSITION FROM WP_Is_Metallic TO WP_Type_Checked
  := WPType_Metallic;
END_TRANSITION
STEP WP_Type_Checked:
  WPTypeChecked(N);
END_STEP
TRANSITION FROM WP_Type_Checked TO Conveyor_ACT_CheckWPType_Init
  := WPTypeChecked;
END_TRANSITION
END_ACTION

ACTION ACT_SortWP:
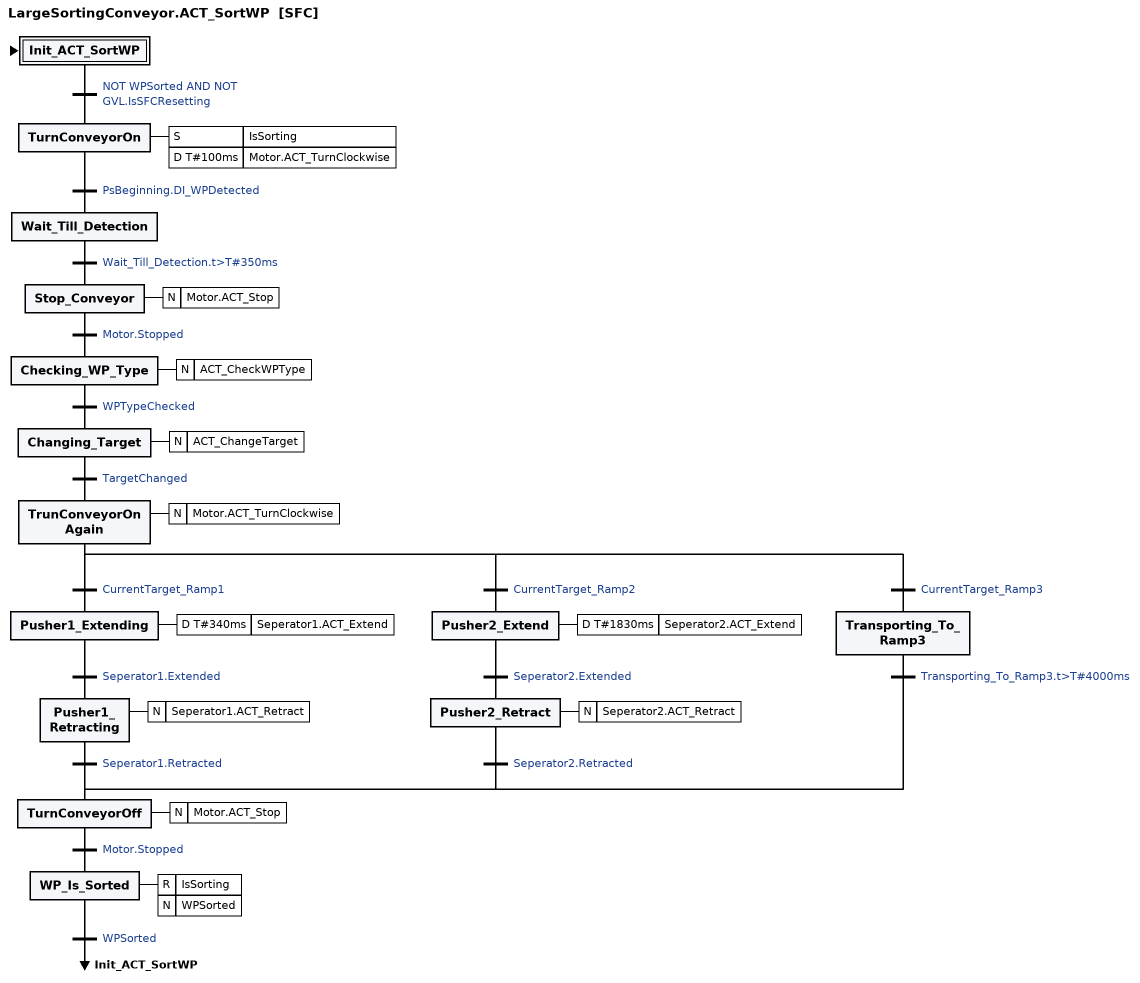
INITIAL_STEP Init_ACT_SortWP:
END_STEP
TRANSITION FROM Init_ACT_SortWP TO TurnConveyorOn
  := NOT WPSorted AND NOT GVL.IsSFCResetting;
END_TRANSITION
STEP TurnConveyorOn:
  IsSorting(S);
  Motor.ACT_TurnClockwise(D, T#100ms);
END_STEP
TRANSITION FROM TurnConveyorOn TO Wait_Till_Detection
  := PsBeginning.DI_WPDetected;
END_TRANSITION
STEP Wait_Till_Detection:
END_STEP
TRANSITION FROM Wait_Till_Detection TO Stop_Conveyor
  := Wait_Till_Detection.t>T#350ms;
END_TRANSITION
STEP Stop_Conveyor:
  Motor.ACT_Stop(N);
END_STEP
TRANSITION FROM Stop_Conveyor TO Checking_WP_Type
  := Motor.Stopped;
END_TRANSITION
STEP Checking_WP_Type:
  ACT_CheckWPType(N);
END_STEP
TRANSITION FROM Checking_WP_Type TO Changing_Target
  := WPTypeChecked;
END_TRANSITION
STEP Changing_Target:
  ACT_ChangeTarget(N);
END_STEP
TRANSITION FROM Changing_Target TO TrunConveyorOnAgain
  := TargetChanged;
END_TRANSITION
STEP TrunConveyorOnAgain:
  Motor.ACT_TurnClockwise(N);
END_STEP
TRANSITION FROM TrunConveyorOnAgain TO Pusher1_Extending
  := CurrentTarget_Ramp1;
END_TRANSITION
TRANSITION FROM TrunConveyorOnAgain TO Pusher2_Extend
  := CurrentTarget_Ramp2;
END_TRANSITION
TRANSITION FROM TrunConveyorOnAgain TO Transporting_To_Ramp3
  := CurrentTarget_Ramp3;
END_TRANSITION
STEP Pusher1_Extending:
  Seperator1.ACT_Extend(D, T#340ms);
END_STEP
TRANSITION FROM Pusher1_Extending TO Pusher1_Retracting
  := Seperator1.Extended;
END_TRANSITION
STEP Pusher1_Retracting:
  Seperator1.ACT_Retract(N);
END_STEP
TRANSITION FROM Pusher1_Retracting TO TurnConveyorOff
  := Seperator1.Retracted;
END_TRANSITION
STEP Pusher2_Extend:
  Seperator2.ACT_Extend(D, T#1830ms);
END_STEP
TRANSITION FROM Pusher2_Extend TO Pusher2_Retract
  := Seperator2.Extended;
END_TRANSITION
STEP Pusher2_Retract:
  Seperator2.ACT_Retract(N);
END_STEP
TRANSITION FROM Pusher2_Retract TO TurnConveyorOff
  := Seperator2.Retracted;
END_TRANSITION
STEP Transporting_To_Ramp3:
END_STEP
TRANSITION FROM Transporting_To_Ramp3 TO TurnConveyorOff
  := Transporting_To_Ramp3.t>T#4000ms;
END_TRANSITION
STEP TurnConveyorOff:
  Motor.ACT_Stop(N);
END_STEP
TRANSITION FROM TurnConveyorOff TO WP_Is_Sorted
  := Motor.Stopped;
END_TRANSITION
STEP WP_Is_Sorted:
  IsSorting(R);
  WPSorted(N);
END_STEP
TRANSITION FROM WP_Is_Sorted TO Init_ACT_SortWP
  := WPSorted;
END_TRANSITION
END_ACTION

ACTION ACT_AutomaticExecute:
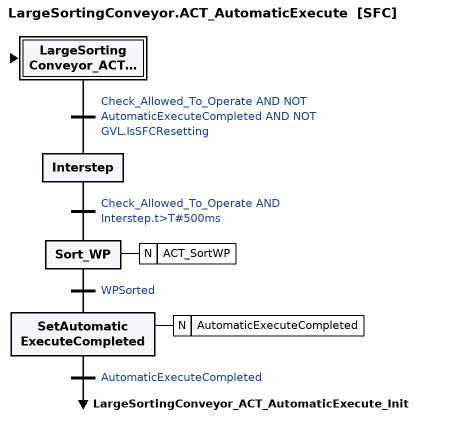
INITIAL_STEP LargeSortingConveyor_ACT_AutomaticExecute_Init:
END_STEP
TRANSITION FROM LargeSortingConveyor_ACT_AutomaticExecute_Init TO Interstep
  := Check_Allowed_To_Operate AND NOT AutomaticExecuteCompleted AND NOT GVL.IsSFCResetting;
END_TRANSITION
STEP Interstep:
END_STEP
TRANSITION FROM Interstep TO Sort_WP
  := Check_Allowed_To_Operate AND Interstep.t>T#500ms;
END_TRANSITION
STEP Sort_WP:
  ACT_SortWP(N);
END_STEP
TRANSITION FROM Sort_WP TO SetAutomaticExecuteCompleted
  := WPSorted;
END_TRANSITION
STEP SetAutomaticExecuteCompleted:
  AutomaticExecuteCompleted(N);
END_STEP
TRANSITION FROM SetAutomaticExecuteCompleted TO LargeSortingConveyor_ACT_AutomaticExecute_Init
  := AutomaticExecuteCompleted;
END_TRANSITION
END_ACTION

ACTION ACT_EmergencyStop:
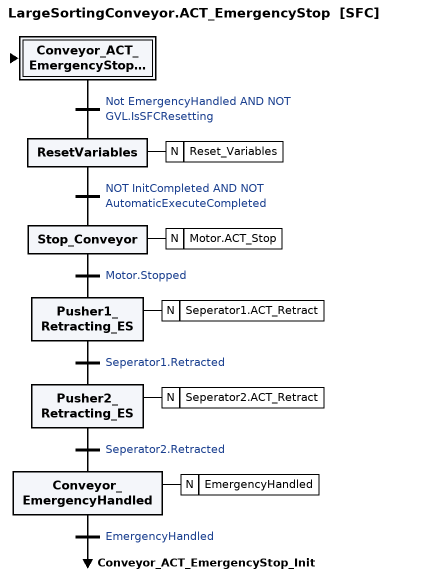
INITIAL_STEP Conveyor_ACT_EmergencyStop_Init:
END_STEP
TRANSITION FROM Conveyor_ACT_EmergencyStop_Init TO ResetVariables
  := Not EmergencyHandled AND NOT GVL.IsSFCResetting;
END_TRANSITION
STEP ResetVariables:
  Reset_Variables(N);
END_STEP
TRANSITION FROM ResetVariables TO Stop_Conveyor
  := NOT InitCompleted AND NOT AutomaticExecuteCompleted;
END_TRANSITION
STEP Stop_Conveyor:
  Motor.ACT_Stop(N);
END_STEP
TRANSITION FROM Stop_Conveyor TO Pusher1_Retracting_ES
  := Motor.Stopped;
END_TRANSITION
STEP Pusher1_Retracting_ES:
  Seperator1.ACT_Retract(N);
END_STEP
TRANSITION FROM Pusher1_Retracting_ES TO Pusher2_Retracting_ES
  := Seperator1.Retracted;
END_TRANSITION
STEP Pusher2_Retracting_ES:
  Seperator2.ACT_Retract(N);
END_STEP
TRANSITION FROM Pusher2_Retracting_ES TO Conveyor_EmergencyHandled
  := Seperator2.Retracted;
END_TRANSITION
STEP Conveyor_EmergencyHandled:
  EmergencyHandled(N);
END_STEP
TRANSITION FROM Conveyor_EmergencyHandled TO Conveyor_ACT_EmergencyStop_Init
  := EmergencyHandled;
END_TRANSITION
END_ACTION

ACTION ACT_Init:
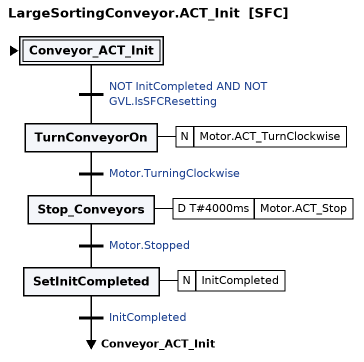
INITIAL_STEP Conveyor_ACT_Init:
END_STEP
TRANSITION FROM Conveyor_ACT_Init TO TurnConveyorOn
  := NOT InitCompleted AND NOT GVL.IsSFCResetting;
END_TRANSITION
STEP TurnConveyorOn:
  Motor.ACT_TurnClockwise(N);
END_STEP
TRANSITION FROM TurnConveyorOn TO Stop_Conveyors
  := Motor.TurningClockwise;
END_TRANSITION
STEP Stop_Conveyors:
  Motor.ACT_Stop(D, T#4000ms);
END_STEP
TRANSITION FROM Stop_Conveyors TO SetInitCompleted
  := Motor.Stopped;
END_TRANSITION
STEP SetInitCompleted:
  InitCompleted(N);
END_STEP
TRANSITION FROM SetInitCompleted TO Conveyor_ACT_Init
  := InitCompleted;
END_TRANSITION
END_ACTION
END_FUNCTION_BLOCK

FUNCTION_BLOCK Stack
VAR_INPUT	
	//Hardware
	Seperator : MonostableCylinder;
	Panel : OperationPanel;	
	WPAvailable : MicroSwitch;
	InductiveSensor : InductiveSensor;
	OpticalSensor : OpticalSensor;
	
	//Software
	StartButton : BOOL;
	InitCompleted : BOOL;
	AutomaticExecuteCompleted : BOOL;
	EmergencyStop : BOOL;
	EmergencyHandled : BOOL;	
	SFCReset : BOOL;	//Only for SFC implementation
END_VAR
VAR_OUTPUT	
	//Software
	WPProvided : BOOL;	
	WPType_White : BOOL;
	WPType_Black : BOOL;
	WPType_Metallic : BOOL;	
END_VAR
VAR	
	//Software
	Timer : TON;
	Check_Crane_PickedUpWp : BOOL;
END_VAR

                  Panel();
StartButton := Panel.StartButton;
EmergencyStop := Panel.EmergencyStop;
Check_Crane_PickedUpWP := Main.Crane_PickedUpStackWP;
                

ACTION Reset_Timer:
                      Timer(IN:=FALSE);
                    
END_ACTION

ACTION Reset_Variables:
                      InitCompleted := FALSE;
AutomaticExecuteCompleted := FALSE;

WPType_White:=FALSE;
WPType_Black:=FALSE;
WPType_Metallic:=FALSE;
                    
END_ACTION

ACTION Set_Timer250ms:
                      Timer(IN:=TRUE, PT:=T#250MS);
                    
END_ACTION

ACTION Set_WPParameters_AND_WPProvided:
                      IF(NOT InductiveSensor.DI_WPMetallic AND NOT OpticalSensor.DI_WPLight)THEN
	WPType_Black:=TRUE;
	WPType_White:=FALSE;
	WPType_Metallic:=FALSE;
ELSIF(NOT InductiveSensor.DI_WPMetallic AND OpticalSensor.DI_WPLight)THEN
	WPType_Black:=FALSE;
	WPType_White:=TRUE;
	WPType_Metallic:=FALSE;
ELSIF(InductiveSensor.DI_WPMetallic)THEN
	WPType_Black:=FALSE;
	WPType_White:=FALSE;
	WPType_Metallic:=TRUE;
END_IF

WPProvided:=TRUE;
                    
END_ACTION

ACTION ACT_ProvideWP:
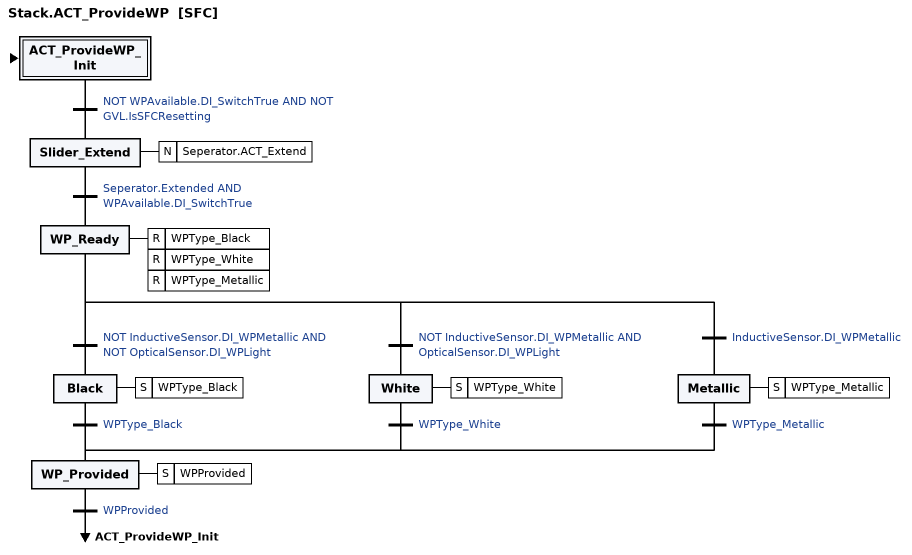
INITIAL_STEP ACT_ProvideWP_Init:
END_STEP
TRANSITION FROM ACT_ProvideWP_Init TO Slider_Extend
  := NOT WPAvailable.DI_SwitchTrue AND NOT GVL.IsSFCResetting;
END_TRANSITION
STEP Slider_Extend:
  Seperator.ACT_Extend(N);
END_STEP
TRANSITION FROM Slider_Extend TO WP_Ready
  := Seperator.Extended AND WPAvailable.DI_SwitchTrue;
END_TRANSITION
STEP WP_Ready:
  WPType_Black(R);
  WPType_White(R);
  WPType_Metallic(R);
END_STEP
TRANSITION FROM WP_Ready TO Black
  := NOT InductiveSensor.DI_WPMetallic AND NOT OpticalSensor.DI_WPLight;
END_TRANSITION
TRANSITION FROM WP_Ready TO White
  := NOT InductiveSensor.DI_WPMetallic AND OpticalSensor.DI_WPLight;
END_TRANSITION
TRANSITION FROM WP_Ready TO Metallic
  := InductiveSensor.DI_WPMetallic;
END_TRANSITION
STEP Black:
  WPType_Black(S);
END_STEP
TRANSITION FROM Black TO WP_Provided
  := WPType_Black;
END_TRANSITION
STEP White:
  WPType_White(S);
END_STEP
TRANSITION FROM White TO WP_Provided
  := WPType_White;
END_TRANSITION
STEP Metallic:
  WPType_Metallic(S);
END_STEP
TRANSITION FROM Metallic TO WP_Provided
  := WPType_Metallic;
END_TRANSITION
STEP WP_Provided:
  WPProvided(S);
END_STEP
TRANSITION FROM WP_Provided TO ACT_ProvideWP_Init
  := WPProvided;
END_TRANSITION
END_ACTION

ACTION ACT_AutomaticExecute:
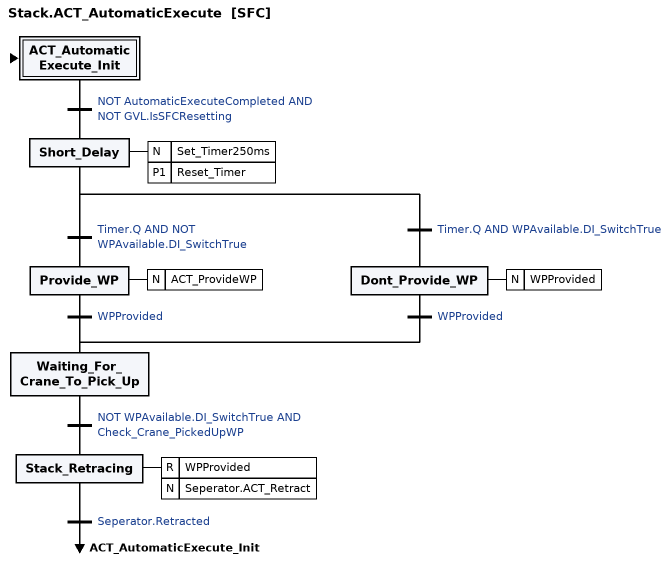
INITIAL_STEP ACT_AutomaticExecute_Init:
END_STEP
TRANSITION FROM ACT_AutomaticExecute_Init TO Short_Delay
  := NOT AutomaticExecuteCompleted AND NOT GVL.IsSFCResetting;
END_TRANSITION
STEP Short_Delay:
  Set_Timer250ms(N);
  Reset_Timer(P1);
END_STEP
TRANSITION FROM Short_Delay TO Provide_WP
  := Timer.Q AND NOT WPAvailable.DI_SwitchTrue;
END_TRANSITION
TRANSITION FROM Short_Delay TO Dont_Provide_WP
  := Timer.Q AND WPAvailable.DI_SwitchTrue;
END_TRANSITION
STEP Provide_WP:
  ACT_ProvideWP(N);
END_STEP
TRANSITION FROM Provide_WP TO Waiting_For_Crane_To_Pick_Up
  := WPProvided;
END_TRANSITION
STEP Dont_Provide_WP:
  WPProvided(N);
END_STEP
TRANSITION FROM Dont_Provide_WP TO Waiting_For_Crane_To_Pick_Up
  := WPProvided;
END_TRANSITION
STEP Waiting_For_Crane_To_Pick_Up:
END_STEP
TRANSITION FROM Waiting_For_Crane_To_Pick_Up TO Stack_Retracing
  := NOT WPAvailable.DI_SwitchTrue AND Check_Crane_PickedUpWP;
END_TRANSITION
STEP Stack_Retracing:
  WPProvided(R);
  Seperator.ACT_Retract(N);
END_STEP
TRANSITION FROM Stack_Retracing TO ACT_AutomaticExecute_Init
  := Seperator.Retracted;
END_TRANSITION
END_ACTION

ACTION ACT_EmergencyStop:
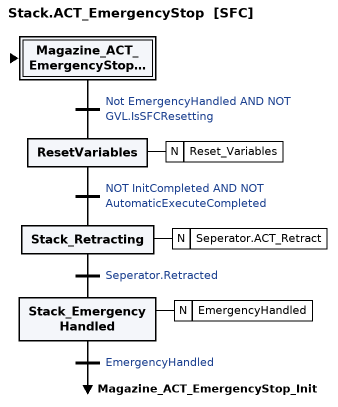
INITIAL_STEP Magazine_ACT_EmergencyStop_Init:
END_STEP
TRANSITION FROM Magazine_ACT_EmergencyStop_Init TO ResetVariables
  := Not EmergencyHandled AND NOT GVL.IsSFCResetting;
END_TRANSITION
STEP ResetVariables:
  Reset_Variables(N);
END_STEP
TRANSITION FROM ResetVariables TO Stack_Retracting
  := NOT InitCompleted AND NOT AutomaticExecuteCompleted;
END_TRANSITION
STEP Stack_Retracting:
  Seperator.ACT_Retract(N);
END_STEP
TRANSITION FROM Stack_Retracting TO Stack_EmergencyHandled
  := Seperator.Retracted;
END_TRANSITION
STEP Stack_EmergencyHandled:
  EmergencyHandled(N);
END_STEP
TRANSITION FROM Stack_EmergencyHandled TO Magazine_ACT_EmergencyStop_Init
  := EmergencyHandled;
END_TRANSITION
END_ACTION

ACTION ACT_Init:
